# EPICS substitutions: db/Beckhoff_9XXX/ecmcEL9410.substitutions
file "ecmcEcSlave.template"
{
  pattern {}
          {}
}

file "ecmcEL9410-chX.template"
{
  pattern {CH_ID}
          {01   }
}
